FUNCTION_BLOCK PUBLIC FB_PiezoDriveDS402CSP EXTENDS FB_PiezoDriveDS402
VAR_INPUT
END_VAR
VAR_OUTPUT
END_VAR
VAR
END_VAR

METHOD Brake : BOOL
SUPER^.Brake();
END_METHOD

METHOD DS402StateMachine
SUPER^.DS402StateMachine();

IF SUPER^.bOperational THEN
	THIS^.HandleMoveRequest();
END_IF
END_METHOD

(*FB_Init is always available implicitly and it is used primarily for initialization.
The return value is not evaluated. For a specific influence, you can also declare the
methods explicitly and provide additional code there with the standard initialization
code. You can evaluate the return value.*)
METHOD FB_Init : BOOL
VAR_INPUT
    (* TRUE: the retain variables are initialized (reset warm / reset cold)*)
    bInitRetains	: BOOL;
    (* TRUE: the instance will be copied to the copy code afterward (online change)   *)
    bInCopyCode	: BOOL;
    stStage : REFERENCE TO  ST_PiezoStage;
END_VAR
END_METHOD

METHOD Halt : BOOL
SUPER^.Halt();
END_METHOD

METHOD HandleMoveRequest
VAR_INPUT
END_VAR
END_METHOD

METHOD Home : BOOL
SUPER^.Home();
END_METHOD

METHOD Interlock : BOOL
SUPER^.Interlock();

// Get a definitive bEnabled reading
CASE SUPER^.stPiezoStage.Axis.Status.MotionState OF
    // We are not enabled if there is an issue
    MC_AXISSTATE_UNDEFINED, MC_AXISSTATE_DISABLED, MC_AXISSTATE_ERRORSTOP:
        SUPER^.stPiezoStage.bEnableDone := FALSE;
    ELSE
        SUPER^.stPiezoStage.bEnableDone := TRUE;
END_CASE
END_METHOD

METHOD Logger : BOOL
SUPER^.Logger();
END_METHOD

METHOD MoveAbsolute
END_METHOD

METHOD MoveRelative : BOOL
END_METHOD

METHOD MoveVelocity : BOOL
END_METHOD


METHOD Power : BOOL
SUPER^.Power();
END_METHOD

METHOD Reset : BOOL
SUPER^.Reset();
END_METHOD

END_FUNCTION_BLOCK

(* stored: Version 1.1.0.1
   POU FB_PiezoDriveDS402CSP: Id {888e3a3f-5a56-4d26-ba78-fe3db55f3f31}, SpecialFunc None
   Method Brake: Id {9a0e88c2-6809-4fed-8bb3-199d998b109d}
   Method DS402StateMachine: Id {73e43dc6-db71-4003-a925-6bc9d3079a38}
   Method FB_Init: Id {600fe1d5-2de2-4cdf-af05-fefe1f75066a}
   Method Halt: Id {749072ab-c58d-463d-9819-0a9dfd276313}
   Method HandleMoveRequest: Id {d7e832c0-06c7-4b10-bdf6-8ebadaa4cbe6}
   Method Home: Id {c98a4912-edf5-4476-8b08-5289494f21e1}
   Method Interlock: Id {1b42e465-3d2a-4756-9fdc-810195b4a90c}
   Method Logger: Id {c96ef2ce-8290-44fd-b101-af264edbe5be}
   Method MoveAbsolute: Id {237c4c50-f769-44ee-a6a5-87a4f79621ba}
   Method MoveRelative: Id {b53079a9-7fd1-49ab-81ed-1d38acd79883}
   Method MoveVelocity: Id {46faa047-3c68-4ca3-a258-bc1a2fc3e753}
   Method Power: Id {28ba770f-aace-4ec5-a43f-418b3d720d89}
   Method Reset: Id {a401ff7f-63d8-4f36-ba52-e017581177a8} *)
